FUNCTION_BLOCK FB_F1Production_SFC EXTENDS FB_Object_Template_SFC
VAR_INPUT
//Discharger
	Discharger_Ready: BOOL;
	Discharger_Done: BOOL;
END_VAR
VAR_OUTPUT
	//Discharger
	Discharger_Execute: BOOL;
	Discharger_Ack: BOOL;
END_VAR
VAR
END_VAR

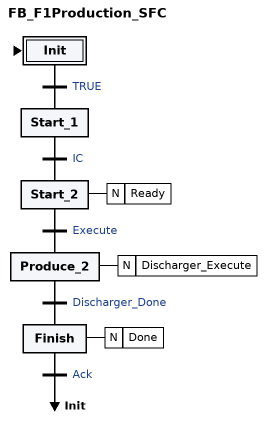
INITIAL_STEP Init:
END_STEP
TRANSITION FROM Init TO Start_1
    := TRUE;
END_TRANSITION
STEP Start_1:
END_STEP
TRANSITION FROM Start_1 TO Start_2
    := IC;
END_TRANSITION
STEP Start_2:
    Ready(N);
END_STEP
TRANSITION FROM Start_2 TO Produce_2
    := Execute;
END_TRANSITION
STEP Produce_2:
    Discharger_Execute(N);
END_STEP
TRANSITION FROM Produce_2 TO Finish
    := Discharger_Done;
END_TRANSITION
STEP Finish:
    Done(N);
END_STEP
TRANSITION FROM Finish TO Init
    := Ack;
END_TRANSITION

END_FUNCTION_BLOCK

(* stored: Version 1.1.0.1, ProductVersion 3.1.4024.6
   POU FB_F1Production_SFC: Id {c71ed4b3-92bb-460f-8f29-6ce922b47ebd}, SpecialFunc None *)
